Yaskawa INFORM job: R1_W29-KM-NOWY-MP.JBI

/JOB
//NAME R1_W29-KM-NOWY-MP
///FOLDERNAME KRIS-SCIANA
//POS
///NPOS 90,90,76,8,0,0
///TOOL 0
///POSTYPE PULSE
///PULSE
C00000=43238,-22106,-75400,-22902,77737,61997
C00001=147206,-70508,-61426,-5078,64470,10052
C00002=131466,-56667,-48515,736,63209,4187
C00003=131466,-54980,-42694,755,60494,4170
C00004=113506,-33390,-29794,19925,71825,-17290
C00005=113506,-33185,-28936,19971,71426,-17358
C00006=113506,-33390,-29794,19925,71825,-17290
C00007=112868,-35881,-31420,20104,71716,-17548
C00008=112868,-35600,-30286,20163,71197,-17638
C00009=113561,-34545,-29600,19989,71140,-17385
C00010=112868,-35758,-30918,20129,71487,-17588
C00011=112868,-36140,-32512,20047,72226,-17461
C00012=136354,-51280,-41701,1511,61812,3408
C00013=136354,-51021,-40811,1517,61397,3403
C00014=136354,-50698,-39732,1523,60899,3397
C00015=136354,-50924,-40485,1518,61246,3402
C00016=136803,-54492,-42487,1355,60638,3567
C00017=136803,-54179,-41498,1361,60192,3562
C00018=136592,-52540,-40585,1438,60472,3485
C00019=136869,-55114,-43142,1328,60719,3595
C00020=144453,-48978,-40378,-1551,62183,6487
C00021=144614,-47865,-39081,-1614,61961,6551
C00022=144614,-47554,-37995,-1619,61451,6556
C00023=144614,-47919,-39277,-1610,62053,6547
C00024=145217,-51071,-41098,-1846,61567,6784
C00025=145217,-50618,-39580,-1859,60864,6795
C00026=144853,-48752,-38502,-1713,61156,6647
C00027=145217,-51290,-41862,-1842,61920,6778
C00028=157952,-17770,-23300,-12207,78345,30733
C00029=158728,-14907,-20947,-12362,78482,30991
C00030=158728,-14691,-19485,-12394,77711,31068
C00031=158728,-14871,-20688,-12368,78345,31004
C00032=160150,-15930,-21486,-12654,78512,31485
C00033=160150,-15709,-20041,-12686,77752,31563
C00034=159415,-15123,-19599,-12539,77666,31315
C00035=160223,-15665,-21406,-12666,78607,31502
C00036=161879,-22396,-36320,-12836,84447,31472
C00037=142488,6488,-14256,2361,98542,-22118
C00038=133363,46753,32411,18168,103839,-75388
C00039=134257,48560,38918,18054,100710,-75538
C00040=135288,45278,34962,18260,101191,-75088
C00041=135288,45576,36212,18216,100605,-75177
C00042=135288,45342,35236,18251,101062,-75107
C00043=135129,48208,38324,18196,100690,-75222
C00044=134852,48929,40025,18108,100106,-75413
C00045=135455,46852,37777,18220,100274,-75167
C00046=134852,48929,40025,18108,100106,-75413
C00047=127142,35538,24761,17068,104170,-77633
C00048=127142,35603,25088,17053,104008,-77655
C00049=127142,35814,26107,17006,103514,-77729
C00050=127142,35603,25088,17053,104008,-77655
C00051=126238,39454,28762,16873,103926,-78000
C00052=125881,39728,30309,16742,103224,-78232
C00053=125732,37660,28163,16737,103501,-78247
C00054=125881,39728,30309,16742,103224,-78232
C00055=118491,40127,27740,15513,106409,-80514
C00056=118491,40543,29820,15420,105379,-80650
C00057=118491,40890,31400,15339,104614,-80747
C00058=118491,40651,30331,15383,105131,-80680
C00059=118523,44303,34188,15348,104645,-80732
C00060=118523,44599,35431,15299,104054,-80808
C00061=118326,42389,33087,15286,104388,-80837
C00062=118523,44599,35431,15299,104054,-80808
C00063=118101,5934,-14778,15437,96959,-81826
C00064=121393,-29214,-36008,9505,78311,-5161
C00065=135587,-47437,-47608,6145,74729,-454
C00066=135289,-41728,-37194,6329,71298,-734
C00067=148370,-34761,-32783,-1982,71305,10330
C00068=156952,-26462,-27171,-12185,75891,24841
C00069=159766,-12029,-16444,-12726,77119,25716
C00070=155246,-26274,-34996,-3885,76881,24554
C00071=111750,-20701,-27381,16937,83641,-24328
C00072=112985,-18825,-21550,16841,80871,-24275
C00073=118829,-29801,-29048,15994,78706,-22486
C00074=124982,-39039,-35244,9713,72691,-11853
C00075=135123,-42276,-37546,5428,70821,-5825
C00076=141350,-43062,-37925,-1384,70008,3170
C00077=141351,-44716,-44807,-1359,73392,3129
C00078=142962,-17764,-29343,-1758,77753,53630
C00079=136048,25534,7501,7664,96790,70217
C00080=129481,57276,49734,18555,109344,89562
C00081=130454,29833,18848,16037,100008,88526
C00082=134058,37987,30412,26327,94520,89687
C00083=134055,36597,23503,26554,97706,90409
C00084=119345,39041,23458,14696,103719,84988
C00085=121095,39149,29000,13196,103006,86871
C00086=134151,53616,46523,11382,106455,85081
C00087=130248,33829,15211,16153,103972,80024
C00088=133531,-22845,-44194,15975,101067,22927
C00089=43238,-22106,-75400,-22902,77737,61997
BC00000=125261,428660,1075156
BC00001=266566,428114,1075173
BC00002=266566,428114,1075173
BC00003=266566,428114,1075173
BC00004=266566,428114,1075173
BC00005=266566,428114,1075173
BC00006=266566,428114,1075173
BC00007=266566,428114,1075173
BC00008=266566,428114,1075173
BC00009=266566,428114,1075173
BC00010=266566,428114,1075173
BC00011=266566,428114,1075173
BC00012=266566,428114,1075173
BC00013=266566,428114,1075173
BC00014=266566,428114,1075173
BC00015=266566,428114,1075173
BC00016=266566,428114,1075173
BC00017=266566,428114,1075173
BC00018=266566,428114,1075173
BC00019=266566,428114,1075173
BC00020=266566,428114,1075173
BC00021=266566,428114,1075173
BC00022=266566,428114,1075173
BC00023=266566,428114,1075173
BC00024=266566,428114,1075173
BC00025=266566,428114,1075173
BC00026=266566,428114,1075173
BC00027=266566,428114,1075173
BC00028=266566,428114,1075173
BC00029=266566,428114,1075173
BC00030=266566,428114,1075173
BC00031=266566,428114,1075173
BC00032=266566,428114,1075173
BC00033=266566,428114,1075173
BC00034=266566,428114,1075173
BC00035=266566,428114,1075173
BC00036=266566,428114,1075173
BC00037=266566,428114,1075173
BC00038=266566,428114,1075173
BC00039=266566,428114,1075173
BC00040=266566,428114,1075173
BC00041=266566,428114,1075173
BC00042=266566,428114,1075173
BC00043=266566,428114,1075173
BC00044=266566,428114,1075173
BC00045=266566,428114,1075173
BC00046=266566,428114,1075173
BC00047=266566,428114,1075173
BC00048=266566,428114,1075173
BC00049=266566,428114,1075173
BC00050=266566,428114,1075173
BC00051=266566,428114,1075173
BC00052=266566,428114,1075173
BC00053=266566,428114,1075173
BC00054=266566,428114,1075173
BC00055=266566,428114,1075173
BC00056=266566,428114,1075173
BC00057=266567,428114,1075172
BC00058=266567,428114,1075172
BC00059=266567,428114,1075172
BC00060=266567,428114,1075172
BC00061=266567,428114,1075172
BC00062=266567,428114,1075172
BC00063=266567,428114,1075172
BC00064=266567,428114,1075172
BC00065=266567,428114,1075172
BC00066=266567,428114,1075172
BC00067=266565,428115,1075170
BC00068=266565,428115,1075170
BC00069=266565,428115,1075168
BC00070=266565,428115,1075170
BC00071=266565,428115,1075170
BC00072=266565,428115,1075170
BC00073=266565,428115,1075170
BC00074=266565,428115,1075170
BC00075=266565,428115,1075170
BC00076=266565,428115,1075170
BC00077=266565,428115,1075170
BC00078=266565,428115,1075170
BC00079=270319,428100,1075172
BC00080=274635,428083,1075174
BC00081=274635,428083,1075174
BC00082=274635,428083,1075174
BC00083=274635,428083,1075174
BC00084=274635,428083,1075174
BC00085=274635,428083,1075174
BC00086=274635,428083,1075174
BC00087=274635,428083,1075174
BC00088=274635,428083,1075174
BC00089=125261,428660,1075156
EC00000=798155,-556476
EC00001=798156,-556476
EC00002=798156,-556476
EC00003=798156,-556476
EC00004=798156,-556476
EC00005=798156,-556476
EC00006=798156,-556476
EC00007=798156,-556476
EC00008=798156,-556476
EC00009=798156,-556476
EC00010=798156,-556476
EC00011=798156,-556476
EC00012=798156,-556476
EC00013=798156,-556476
EC00014=798156,-556476
EC00015=798156,-556476
EC00016=798156,-556476
EC00017=798156,-556476
EC00018=798156,-556476
EC00019=798156,-556476
EC00020=798156,-556476
EC00021=798156,-556476
EC00022=798156,-556476
EC00023=798156,-556476
EC00024=798156,-556476
EC00025=798156,-556476
EC00026=798156,-556476
EC00027=798156,-556476
EC00028=798156,-556476
EC00029=798156,-556476
EC00030=798156,-556476
EC00031=798156,-556476
EC00032=798156,-556476
EC00033=798156,-556476
EC00034=798156,-556476
EC00035=798156,-556476
EC00036=798156,-556476
EC00037=798156,-556476
EC00038=798156,-556476
EC00039=798156,-556476
EC00040=798156,-556476
EC00041=798156,-556476
EC00042=798156,-556476
EC00043=798156,-556476
EC00044=798156,-556476
EC00045=798154,-556476
EC00046=798154,-556476
EC00047=798154,-556476
EC00048=798154,-556476
EC00049=798154,-556476
EC00050=798154,-556476
EC00051=798154,-556476
EC00052=798154,-556476
EC00053=798151,-556476
EC00054=798151,-556476
EC00055=798147,-556476
EC00056=798151,-556476
EC00057=798151,-556476
EC00058=798151,-556476
EC00059=798151,-556476
EC00060=798151,-556476
EC00061=798151,-556476
EC00062=798151,-556476
EC00063=798151,-556476
EC00064=798151,-556476
EC00065=798154,-556476
EC00066=798156,-556476
EC00067=798156,-556476
EC00068=798156,-556476
EC00069=798156,-556476
EC00070=798156,-556476
EC00071=798156,-556476
EC00072=798156,-556476
EC00073=798156,-556476
EC00074=798156,-556476
EC00075=798155,-556476
///POSTYPE BASE
///RECTAN
///RCONF 0,0,0,0,1,0,0,0,0,0,0,0,0,0,0,0,0,0,0,0,0,0,0,0
P00006=2.006,1.622,-0.565,0.0000,0.0000,0.0000
P00021=0.073,2.058,-0.109,0.0000,0.0000,0.0000
P00022=2.006,1.622,-0.565,0.0000,0.0000,0.0000
///RCONF 0,0,0,0,0,0,0,0,0,0,0,0,0,0,0,0,0,0,0,0,0,0,0,0
P00023=-2.957,-4.083,2.762,0.0000,0.0000,0.0000
P00024=-1.466,-0.226,-0.419,0.0000,0.0000,0.0000
P00025=3.643,0.007,-2.585,0.0000,0.0000,0.0000
P00026=2.644,0.055,-2.583,0.0000,0.0000,0.0000
P00027=2.278,0.099,-4.210,0.0000,0.0000,0.0000
//INST
///DATE 2024/12/27 10:42
///ATTR SC,RW
///GROUP1 RB1,BS1
///GROUP2 ST1
NOP
SFTOF
MOVJ C00000 BC00000 VJ=15.00  +MOVJ EC00000 VJ=15.00
MOVJ C00001 BC00001 VJ=50.00  +MOVJ EC00001 VJ=50.00
MOVJ C00002 BC00002 VJ=15.00  +MOVJ EC00002 VJ=15.00
'SEARCH
MOVL C00003 BC00003 V=58.3  +MOVJ EC00003 VJ=15.00
MOVL C00004 BC00004 V=58.3  +MOVJ EC00004 VJ=15.00
REFP 3 RB1 C00005 BC00005
CALL JOB:SEARCH-R1
SET P021 P006
SFTON P021
MOVL C00006 BC00006 V=58.3  +MOVJ EC00005 VJ=15.00
MOVL C00007 BC00007 V=83.3  +MOVJ EC00006 VJ=15.00
MOVL C00008 BC00008 V=83.3  +MOVJ EC00007 VJ=15.00
REFP 3 RB1 C00009 BC00009
CALL JOB:SEARCH-R1
SET P021 P006
SFTON P021
MOVL C00010 BC00010 V=58.3  +MOVJ EC00008 VJ=15.00
MOVL C00011 BC00011 V=100.0  +MOVJ EC00009 VJ=15.00
SFTOF
MOVL C00012 BC00012 V=133.3  +MOVJ EC00010 VJ=15.00
MOVL C00013 BC00013 V=58.3  +MOVJ EC00011 VJ=15.00
REFP 3 RB1 C00014 BC00014
CALL JOB:SEARCH-R1
SET P022 P006
SFTON P022
MOVL C00015 BC00015 V=58.3  +MOVJ EC00012 VJ=15.00
MOVL C00016 BC00016 V=100.0  +MOVJ EC00013 VJ=15.00
MOVL C00017 BC00017 V=100.0  +MOVJ EC00014 VJ=15.00
REFP 3 RB1 C00018 BC00018
CALL JOB:SEARCH-R1
SET P022 P006
SFTON P022
MOVL C00019 BC00019 V=100.0  +MOVJ EC00015 VJ=15.00
SFTOF
MOVL C00020 BC00020 V=166.7  +MOVJ EC00016 VJ=15.00
MOVL C00021 BC00021 V=58.3  +MOVJ EC00017 VJ=15.00
REFP 3 RB1 C00022 BC00022
CALL JOB:SEARCH-R1
SET P023 P006
SFTON P023
MOVL C00023 BC00023 V=58.3  +MOVJ EC00018 VJ=15.00
MOVL C00024 BC00024 V=83.3  +MOVJ EC00019 VJ=15.00
MOVL C00025 BC00025 V=83.3  +MOVJ EC00020 VJ=15.00
REFP 3 RB1 C00026 BC00026
CALL JOB:SEARCH-R1
SET P023 P006
SFTON P023
MOVL C00027 BC00027 V=100.0  +MOVJ EC00021 VJ=15.00
MOVL C00028 BC00028 V=100.0  +MOVJ EC00022 VJ=15.00
SFTOF
MOVL C00029 BC00029 V=58.3  +MOVJ EC00023 VJ=15.00
REFP 3 RB1 C00030 BC00030
CALL JOB:SEARCH-R1
SET P024 P006
SFTON P024
MOVL C00031 BC00031 V=58.3  +MOVJ EC00024 VJ=15.00
MOVL C00032 BC00032 V=100.0  +MOVJ EC00025 VJ=15.00
MOVL C00033 BC00033 V=100.0  +MOVJ EC00026 VJ=15.00
REFP 3 RB1 C00034 BC00034
CALL JOB:SEARCH-R1
SET P024 P006
SFTON P024
MOVL C00035 BC00035 V=100.0  +MOVJ EC00027 VJ=15.00
SSFTOF
MOVJ C00036 BC00036 VJ=100.00  +MOVJ EC00028 VJ=100.00
MOVJ C00037 BC00037 VJ=100.00  +MOVJ EC00029 VJ=100.00
MOVJ C00038 BC00038 VJ=100.00  +MOVJ EC00030 VJ=100.00
MOVL C00039 BC00039 V=166.7  +MOVJ EC00031 VJ=15.00
MOVL C00040 BC00040 V=58.3  +MOVJ EC00032 VJ=15.00
REFP 3 RB1 C00041 BC00041
CALL JOB:SEARCH-R1
SET P025 P006
SFTON P025
MOVL C00042 BC00042 V=58.3  +MOVJ EC00033 VJ=15.00
MOVL C00043 BC00043 V=100.0  +MOVJ EC00034 VJ=15.00
MOVL C00044 BC00044 V=100.0  +MOVJ EC00035 VJ=15.00
REFP 3 RB1 C00045 BC00045
CALL JOB:SEARCH-R1
SET P025 P006
SFTON P025
MOVL C00046 BC00046 V=100.0  +MOVJ EC00036 VJ=15.00
SSFTOF
MOVL C00047 BC00047 V=250.0  +MOVJ EC00037 VJ=100.00
MOVL C00048 BC00048 V=58.3  +MOVJ EC00038 VJ=15.00
REFP 3 RB1 C00049 BC00049
CALL JOB:SEARCH-R1
SET P026 P006
SFTON P026
MOVL C00050 BC00050 V=58.3  +MOVJ EC00039 VJ=15.00
MOVL C00051 BC00051 V=100.0  +MOVJ EC00040 VJ=15.00
MOVL C00052 BC00052 V=100.0  +MOVJ EC00041 VJ=15.00
REFP 3 RB1 C00053 BC00053
CALL JOB:SEARCH-R1
SET P026 P006
SFTON P026
MOVL C00054 BC00054 V=100.0  +MOVJ EC00042 VJ=15.00
MOVL C00055 BC00055 V=250.0  +MOVJ EC00043 VJ=100.00
MOVL C00056 BC00056 V=58.3  +MOVJ EC00044 VJ=15.00
REFP 3 RB1 C00057 BC00057
CALL JOB:SEARCH-R1
SET P027 P006
SFTON P027
MOVL C00058 BC00058 V=58.3  +MOVJ EC00045 VJ=15.00
MOVL C00059 BC00059 V=100.0  +MOVJ EC00046 VJ=15.00
MOVL C00060 BC00060 V=100.0  +MOVJ EC00047 VJ=15.00
REFP 3 RB1 C00061 BC00061
CALL JOB:SEARCH-R1
SET P027 P006
SFTON P027
MOVL C00062 BC00062 V=100.0  +MOVJ EC00048 VJ=15.00
SFTOF
MOVJ C00063 BC00063 VJ=100.00  +MOVJ EC00049 VJ=100.00
MOVJ C00064 BC00064 VJ=100.00  +MOVJ EC00050 VJ=100.00
MOVJ C00065 BC00065 VJ=100.00  +MOVJ EC00051 VJ=100.00
CALL JOB:COFNIJ_DRUT
SFTON P023
MOVL C00066 BC00066 V=100.0 PL=0  +MOVJ EC00052 VJ=15.00
MACRO1 MJ#(0) ARGF7
ARCON
MOVL C00067 BC00067 V=10.8  +MOVJ EC00053 VJ=15.00
MOVL C00068 BC00068 V=10.8  +MOVJ EC00054 VJ=15.00
SSFTON P024
MOVL C00069 BC00069 V=10.8  +MOVJ EC00055 VJ=15.00
ARCOF
SFTOF
MOVJ C00070 BC00070 VJ=30.00  +MOVJ EC00056 VJ=15.00
MOVJ C00071 BC00071 VJ=100.00  +MOVJ EC00057 VJ=100.00
SFTOF
SFTON P021
MOVL C00072 BC00072 V=100.0 PL=0  +MOVJ EC00058 VJ=15.00
ARCON
MOVL C00073 BC00073 V=10.8  +MOVJ EC00059 VJ=15.00
MOVL C00074 BC00074 V=10.8  +MOVJ EC00060 VJ=15.00
SFTON P022
MOVL C00075 BC00075 V=10.8  +MOVJ EC00061 VJ=15.00
MOVL C00076 BC00076 V=10.8  +MOVJ EC00062 VJ=15.00
ARCOF
MOVJ C00077 BC00077 VJ=15.00  +MOVJ EC00063 VJ=15.00
SFTOF
MOVJ C00078 BC00078 VJ=100.00  +MOVJ EC00064 VJ=100.00
MOVJ C00079 BC00079 VJ=100.00  +MOVJ EC00065 VJ=100.00
MOVJ C00080 BC00080 VJ=50.00  +MOVJ EC00066 VJ=50.00
SFTOF
SFTON P026
MOVL C00081 BC00081 V=250.0 PL=0  +MOVJ EC00067 VJ=15.00
ARCON
SFTON P025
MOVL C00082 BC00082 V=10.8  +MOVJ EC00068 VJ=15.00
ARCOF
MOVJ C00083 BC00083 VJ=15.00  +MOVJ EC00069 VJ=15.00
SFTOF
MOVJ C00084 BC00084 VJ=15.00  +MOVJ EC00070 VJ=15.00
SFTON P027
MOVL C00085 BC00085 V=100.0 PL=0  +MOVJ EC00071 VJ=15.00
ARCON
SFTON P026
MOVL C00086 BC00086 V=10.8  +MOVJ EC00072 VJ=15.00
ARCOF
SFTOF
MOVJ C00087 BC00087 VJ=15.00  +MOVJ EC00073 VJ=15.00
MOVJ C00088 BC00088 VJ=100.00  +MOVJ EC00074 VJ=100.00
MOVJ C00089 BC00089 VJ=100.00  +MOVJ EC00075 VJ=20.00
SFTOF
END
